// TIA Portal V18 export
TYPE "SubProcessParameterP040_ShW"
// stored: IsFailsafeCompliant false
   STRUCT
      SubProcessParameter : Struct
         leaktest_p1 : Struct
            leaktest_p1_value : Real;
            leaktest_p1_result : Int;
            leaktest_p1_NG_code : String[9];
         END_STRUCT;
         leaktest_p2 : Struct
            leaktest_p2_value : Real;
            leaktest_p2_result : Int;
            leaktest_p2_NG_code : String[9];
         END_STRUCT;
      END_STRUCT;
   END_STRUCT;
END_TYPE
